FUNCTION_BLOCK FB_EventF2
VAR_INPUT
	FB_Bacnet : FB_BACnet_DAIKIN_MasterStation_III_No_1;
END_VAR
VAR_OUTPUT
	sDebug : STRING(200);
END_VAR
VAR
	fbMsg : FB_TcMessage;
	aUnits : ARRAY[1..23] OF AC_Unit_Status;
	stUnit   : AC_Unit_Status;
	i: INT;
	sMsgText: STRING;
END_VAR
VAR RETAIN
	aPrevState : ARRAY[1..23] OF BOOL := [FALSE(*23*)];
END_VAR


aUnits[1].bPresVal := FB_Bacnet.StartStopStatus_128.bPresVal;
aUnits[1].sUnitName := 'F2-1 (1-00)';
aUnits[2].bPresVal := FB_Bacnet.StartStopStatus_129.bPresVal;
aUnits[2].sUnitName := 'F2-2 (1-01)';
aUnits[3].bPresVal := FB_Bacnet.StartStopStatus_130.bPresVal;
aUnits[3].sUnitName := 'F2-3 (1-02)';
aUnits[4].bPresVal := FB_Bacnet.StartStopStatus_131.bPresVal;
aUnits[4].sUnitName := 'F2-4 (1-03)';
aUnits[5].bPresVal := FB_Bacnet.StartStopStatus_132.bPresVal;
aUnits[5].sUnitName := 'F2-5 (1-04)';
aUnits[6].bPresVal := FB_Bacnet.StartStopStatus_133.bPresVal;
aUnits[6].sUnitName := 'F2-6 (1-05)';
aUnits[7].bPresVal := FB_Bacnet.StartStopStatus_134.bPresVal;
aUnits[7].sUnitName := 'F2-7 (1-06)';
aUnits[8].bPresVal := FB_Bacnet.StartStopStatus_135.bPresVal;
aUnits[8].sUnitName := 'F2-8 (1-07)';
aUnits[9].bPresVal := FB_Bacnet.StartStopStatus_136.bPresVal;
aUnits[9].sUnitName := 'F2-9 (1-08)';
aUnits[10].bPresVal := FB_Bacnet.StartStopStatus_137.bPresVal;
aUnits[10].sUnitName := 'F2-10 (1-09)';
aUnits[11].bPresVal := FB_Bacnet.StartStopStatus_138.bPresVal;
aUnits[11].sUnitName := 'F2-11 (1-10)';
aUnits[12].bPresVal := FB_Bacnet.StartStopStatus_139.bPresVal;
aUnits[12].sUnitName := 'F2-12 (1-11)';
//aUnits[13].bPresVal := FB_Bacnet.StartStopStatus_140.bPresVal;
//aUnits[13].sUnitName := 'F2-13 (1-12)';
aUnits[14].bPresVal := FB_Bacnet.StartStopStatus_141.bPresVal;
aUnits[14].sUnitName := 'F2-14 (1-13)';
aUnits[15].bPresVal := FB_Bacnet.StartStopStatus_142.bPresVal;
aUnits[15].sUnitName := 'F2-15 (1-14)';
aUnits[16].bPresVal := FB_Bacnet.StartStopStatus_143.bPresVal;
aUnits[16].sUnitName := 'F2-16 (1-15)';
aUnits[17].bPresVal := FB_Bacnet.StartStopStatus_144.bPresVal;
aUnits[17].sUnitName := 'F2-17 (2-00)';
aUnits[18].bPresVal := FB_Bacnet.StartStopStatus_145.bPresVal;
aUnits[18].sUnitName := 'F2-18 (2-01)';
aUnits[19].bPresVal := FB_Bacnet.StartStopStatus_146.bPresVal;
aUnits[19].sUnitName := 'F2-19 (2-02)';
aUnits[20].bPresVal := FB_Bacnet.StartStopStatus_147.bPresVal;
aUnits[20].sUnitName := 'F2-20 (2-03)';
aUnits[21].bPresVal := FB_Bacnet.StartStopStatus_148.bPresVal;
aUnits[21].sUnitName := 'F2-21 (2-04)';
aUnits[22].bPresVal := FB_Bacnet.StartStopStatus_176.bPresVal;
aUnits[22].sUnitName := 'F2-IT-1 (4-00)';
//aUnits[23].bPresVal := FB_Bacnet.StartStopStatus_177.bPresVal;
//aUnits[23].sUnitName := 'F2-IT-2 (4-01)';

FOR i := 1 TO 23 DO
    stUnit := aUnits[i];

    // Detect ON/OFF state change
    IF aUnits[i].bPresVal <> aPrevState[i] THEN
        // --------------------------------------------------------
        // (a) Send TwinCAT message as before
        // --------------------------------------------------------
        IF aUnits[i].bPresVal THEN
            sMsgText := CONCAT(stUnit.sUnitName, ' is Turned ON');
        ELSE
            sMsgText := CONCAT(stUnit.sUnitName, ' is Turned OFF');
        END_IF

        fbMsg.CreateEx(TC_EVENTS.UnitPowerStatus.EventPowerStatus, 0);
        fbMsg.ipArguments.AddString(sMsgText);
        fbMsg.Send(0);

        // --------------------------------------------------------
        // (b) Push event to global CSV queue (for P_CSVWrite_TextMode)
        // --------------------------------------------------------
        IF g_iCount < g_CSV_BUF_SIZE THEN
            g_aUnitName[g_iWriteIdx] := stUnit.sUnitName;
            g_aState[g_iWriteIdx]    := aUnits[i].bPresVal;
            g_iWriteIdx := g_iWriteIdx + 1;
            IF g_iWriteIdx > g_CSV_BUF_SIZE THEN g_iWriteIdx := 1; END_IF
            g_iCount := g_iCount + 1;
        END_IF

        // --------------------------------------------------------
        // (c) Update previous state
        // --------------------------------------------------------
        aPrevState[i] := aUnits[i].bPresVal;
    END_IF
END_FOR

// ------------------------------------------------------------
// Optional debug info
// ------------------------------------------------------------
sDebug := CONCAT('Queued=', INT_TO_STRING(g_iCount));

END_FUNCTION_BLOCK

(* stored: Version 1.1.0.1, ProductVersion 3.1.4024.14
   POU FB_EventF2: Id {8ee617d1-75f4-470f-b752-e85ad461cd13}, SpecialFunc None *)
